Fanuc KAREL source: kt00071.KL

-- PROVISIONAL review KL for V770-1; original PC SHA256 6d72389978284004f0d60af71be8d8c44c78dd57799b70084347fddd6cd1fcb3
-- Incomplete behavior may be omitted. Consult companion uncertainty JSON. Do not deploy.
PROGRAM KT00071
%NOLOCKGROUP
VAR
  I1 : INTEGER
  OUT : INTEGER
-- UNRESOLVED_DECL H2 type=002017
BEGIN
  -- UNRESOLVED_PC offsets 5-16; opcodes 2E,23
  -- UNRESOLVED_PC offsets 21-35; opcodes 2E,22,9D,33,B4
  -- UNRESOLVED_PC offsets 40-62; opcodes 21,22,9D,33,B3,54,23
  -- UNRESOLVED_PC offsets 67-71; opcodes 7F
END KT00071
